PROGRAM PRGCompilation
VAR
	fbLogger						: FB_BaseLogger;
	fbMachineControl				: FB_MCMachineControl;
	fbMachineControlHMIConnector	: FB_MCHMIMachineControl_HMI (
										itfBaseLoggerConnector		:= fbLogger,
	                                    itfMachineControlConnector	:= fbMachineControl
									);
END_VAR

END_PROGRAM

(* stored: Version 1.1.0.1
   POU PRGCompilation: Id {6da300e2-4a5f-4e8e-a9ba-b4f69f4dff67}, SpecialFunc None *)
